PROGRAM MAIN
VAR
END_VAR

END_PROGRAM

(* stored: Version 1.1.0.1, ProductVersion 3.1.0.26
   POU MAIN: Id {27968eaf-cc56-466e-9fb5-48fcdcc10757} *)
